TYPE sCCDataStreamSetup :
STRUCT
	byBlockType: BYTE;
	byBlockLength: BYTE;
	byFillByte1: BYTE;
	byFillByte2: BYTE;
	bySelectTrack: BYTE;
	bySelectAxis: BYTE;
	bySelectSignal: BYTE;
	bySelectFlag: BYTE;
END_STRUCT
END_TYPE

(* stored: Version 1.1.0.1, ProductVersion 3.1.4022.16
   DUT sCCDataStreamSetup: Id {681e34af-7d57-46c7-9cae-fe6a1b2b3f49} *)
